// TIA Portal V20 export
TYPE "NDD_Ordenes"
   STRUCT
      Operacion_EntradaPaleta : Bool;
      Operacion_PaletizarPaleta : Bool;
      Operacion_EvacuarPaleta : Bool;
      Operacion_TElev_Garras : Bool;
      Operacion_TElev_Horquilla : Bool;
      Operacion_Horq_Garra : Bool;
      Operacion_Garra_Elev : Bool;
      Libre_07 : Bool;
      TElev_PaletaVacia : Bool;
      TElev_PaletaCargada : Bool;
      TElev_Enfradar : Bool;
      TElev_Paletizar : Bool;
      Libre_13 : Bool;
      Libre_14 : Bool;
      Libre_15 : Bool;
      TElev_SinUT : Bool;
      TElev_CodigoEnfardado : Int;
      TElev_CotaAltura : Int;
   END_STRUCT;
END_TYPE
